PROGRAM MAIN
VAR
	generatePDF : BOOL;
	myData : MyData;
	pdfReport : PDFReport;
END_VAR

// To run the demo you will need the following
//
// 1) you are running the mobject companion app, mobject-app
// 2) you have copied the pdfReport folder in to the mobject app's extensions folder
// 3) you have copied template.json to C:\temp\

IF generatePDF THEN
	generatePDF := FALSE;
	pdfReport.Generate(
		SourceData := myData,
		TemplateName := 'C:\temp\template.json',
		FileName := 'test.pdf',
		FilePath := 'C:\temp\'
	);
END_IF

IF pdfReport.Busy THEN
	pdfReport.CyclicCall();
END_IF

END_PROGRAM

(* stored: Version 1.1.0.1, ProductVersion 3.1.4024.12
   POU MAIN: Id {ca1e1f26-6d15-4483-9500-7f4e2de7b73c}, SpecialFunc None *)
